# EPICS autosave request: ADBruker/iocs/brukerIOC/iocBoot/iocBruker/auto_settings.req
file "BIS_settings.req",          P=$(P),  R=cam1:
ffile "NDStdArrays_settings.req", P=$(P),  R=image1:
file "commonPlugin_settings.req", P=$(P)
